(* PLC project bottle, Dassault Systèmes ControlBuild 2024x *)
(* stored: creationDateTime 2023-10-03T11:13:40-01:00 *)

FUNCTION_BLOCK bottling_line.bottle
  VAR_INPUT
    pulseGenerator : BOOL := false;
    loading : BOOL := false;
    evacuation : BOOL := false;
    inputFlow : REAL := 0.0;
  END_VAR
  VAR_OUTPUT
    bottleFilled : BOOL := false;
    bottlePresent : BOOL := false;
  END_VAR
  VAR
    existenceOfBottle1 : BOOL := false;
    existenceOfBottle2 : BOOL := false;
    existenceOfBottle3 : BOOL := false;
    levelOfBottle1 : REAL := 0.0;
    levelOfBottle2 : REAL := 0.0;
    levelOfBottle3 : REAL := 0.0;
    positionOfBottle1 : DINT := 0;
    positionOfBottle2 : DINT := 0;
    positionOfBottle3 : DINT := 0;
    edge_loading : BOOL := false;
    edge_evacuation : BOOL := false;
    edge_pulseGenerator : BOOL := false;
    first : BOOL := true;
  END_VAR
  VAR CONSTANT
    maxLevel : REAL := 100.0;
    increment : INT := 1;
  END_VAR


ACTION C_source_code:
/* Arrival of a bottle on the conveyor belt			*/
/* -------------------------------------------------------------------------------------------	*/
if(first) {
	edge_loading = loading;
	edge_evacuation = evacuation;
	edge_pulseGenerator = pulseGenerator;
	first = 0;
}
if (loading > edge_loading)
     if (! existenceOfBottle1) 
          {
          existenceOfBottle1=1;
          positionOfBottle1=0;
          }
     else 
          if (! existenceOfBottle2) 
               {
               existenceOfBottle2=1;
               positionOfBottle2=0;
               }
          else 
               if (! existenceOfBottle3) 
                    {
                    existenceOfBottle3=1;
                    positionOfBottle3=0;
                    }


/* Evacuation of a bottle at the end of the conveyor belt	*/
/* -------------------------------------------------------------------------------------------	*/
if (evacuation > edge_evacuation)
     {
     if (existenceOfBottle1 && (positionOfBottle1 >= 20)) 
          {
          existenceOfBottle1=0;
          levelOfBottle1=0;
          }
     if (existenceOfBottle2 && (positionOfBottle2 >= 20)) 
          {
          existenceOfBottle2=0;
          levelOfBottle2=0;
          }
     if (existenceOfBottle3 && (positionOfBottle3 >= 20)) 
          {
          existenceOfBottle3=0;
          levelOfBottle3=0;
          }
     }


/* Movement of the bottles on the conveyor			*/
/* -------------------------------------------------------------------------------------------	*/
if (pulseGenerator > edge_pulseGenerator)
     {
     if existenceOfBottle1 positionOfBottle1=positionOfBottle1+increment;
     if existenceOfBottle2 positionOfBottle2=positionOfBottle2+increment;
     if existenceOfBottle3 positionOfBottle3=positionOfBottle3+increment;
      }

/* Detection of a bottle in the filling area			*/
/* --------------------------------------------------------------------------------------------	*/
if (existenceOfBottle1 && (positionOfBottle1 >=10) && (positionOfBottle1 <= 15)) 
     {
     bottlePresent=1;
     levelOfBottle1=levelOfBottle1+inputFlow;
     if (levelOfBottle1 >= maxLevel) 
          {
          bottleFilled=1;
          levelOfBottle1=maxLevel;
          }
     else bottleFilled=0;
     }
else
     if (existenceOfBottle2 && (positionOfBottle2 >=10) && (positionOfBottle2 <= 15)) 
          {
          bottlePresent=1;
          levelOfBottle2=levelOfBottle2+inputFlow;
          if (levelOfBottle2 >= maxLevel) 
          {
               bottleFilled=1;
               levelOfBottle2=maxLevel;
               }
          else bottleFilled=0;
          }
     else
          if (existenceOfBottle3 && (positionOfBottle3 >=10) && (positionOfBottle3 <= 15)) 
               {
               bottlePresent=1;
               levelOfBottle3=levelOfBottle3+inputFlow;
               if (levelOfBottle3 >= maxLevel) 
                    {
                   bottleFilled=1;
                   levelOfBottle3=maxLevel;
                   }
               else bottleFilled=0;
               }
          else bottlePresent=0;

edge_loading = loading;
edge_evacuation = evacuation;
edge_pulseGenerator = pulseGenerator;
END_ACTION
END_FUNCTION_BLOCK
